(* CODESYS project tcl_simpleunittestlibrary.library
   Company: Red Rock Controls Limited
   Description: ClearTests() added to TTestRunner
   Version: 1.0.7.0
   Placeholder: tcl_SimpleUnitTestLibrary
   Author: Roger Christopher
   Title: tcl_SimpleUnitTestLibrary

Project tree, tasks and I/O mapping:
  libraries: Tc2_EtherCAT, * (Beckhoff Automation GmbH); Tc2_Standard, * (Beckhoff Automation GmbH); Tc2_System, * (Beckhoff Automation GmbH); Tc2_Utilities, * (Beckhoff Automation GmbH); Tc3_DynamicMemory, * (Beckhoff Automation GmbH); Tc3_Module, * (Beckhoff Automation GmbH); tcl_StringUtils, * (Red Rock Controls Limited)
  DUTs/
    data type TTestResult
  GVLs/
    global variables Parameters
    global variables TestFramework
  Unit Test Framework/
    Assertions/
      interface IAssertionMessageList: AddMessage, Clear
      function block TAssertion [ST]: AssertEquals_BLOB, AssertEquals_BOOL, AssertEquals_BYTE, AssertEquals_DINT, AssertEquals_DWORD, AssertEquals_INT, AssertEquals_INTERFACE, AssertEquals_LINT, AssertEquals_LREAL, AssertEquals_PVOID, AssertEquals_REAL, AssertEquals_STRING, AssertEquals_UDINT, AssertEquals_UINT, AssertEquals_ULINT, AssertEquals_WORD, FB_init, AssertionFailed, AssertionMessage
    Message list/
      function block TAssertionMessageList [ST]: AddMessage, Clear
    Test Runner/
      Test Runner/
        function block TTestRunner [ST]: AddTest, AddTestSuite, ClearResults, ClearTests, getTimeStampAsString, Results, TestCount, TestsRunning
    TestSuite/
      interface ITestSuite: AddTest, GetTest, Name, TestCount
      function block TTestSuite [ST]: AddTest, FB_init, GetTest, Name, TestCount
    Unit Test/
      interface IAssertionListener: OnAssertionFailed, TestName
      interface IUnitTest: Execute, Initialise, TestHasFailed, TestHasFinished, TestName
      function block TUnitTestBase [ST]: Execute, FB_init, Initialise, OnAssertionFailed, setTestName, TestFinished, TestHasFailed, TestHasFinished, TestName
  Version/
    global variables Global_Version
  VISUs/
    visualisation Visualization
  GlobalImagePool
  00000000-0000-0000-0000-000000000000|Images\Failed.png
  00000000-0000-0000-0000-000000000000|Images\Passed.png
  00000000-0000-0000-0000-000000000000|Images\BlueRight.png
  text list GlobalTextList
*)

// DUTs/TTestResult
TYPE TTestResult :
STRUCT
    TestName         : T_MaxString;
    TestState        : T_MaxString;
    ImageRef         : T_MaxString;
    TestCompleteTime : T_MaxString;
END_STRUCT
END_TYPE

// GVLs/Parameters
VAR_GLOBAL CONSTANT
    MAX_TESTS              : DINT := 200;
    MAX_ASSERTION_MESSAGES : DINT := 200;
END_VAR

// GVLs/TestFramework
{attribute 'qualified_only'}
VAR_GLOBAL
    TestRunner : TTestRunner;
END_VAR

// Version/Global_Version
{attribute 'TcGenerated'}
{attribute 'no-analysis'}
{attribute 'linkalways'}
// This function has been automatically generated from the project information.
VAR_GLOBAL CONSTANT
	{attribute 'const_non_replaced'}
	stLibVersion_tcl_SimpleUnitTestLibrary : ST_LibVersion := (iMajor := 1, iMinor := 0, iBuild := 7, iRevision := 0, nFlags := 0, sVersion := '1.0.7.0');
END_VAR

// Unit Test Framework/Assertions/IAssertionMessageList
INTERFACE IAssertionMessageList

METHOD AddMessage : BOOL
VAR_INPUT
    Message : T_MaxString;
END_VAR
END_METHOD

METHOD Clear
VAR_INPUT
END_VAR
END_METHOD

END_INTERFACE

// Unit Test Framework/Assertions/TAssertion
FUNCTION_BLOCK TAssertion
VAR_INPUT
END_VAR
VAR_OUTPUT
END_VAR
VAR
    _AssertionFailed : BOOL;
    _AssertionMessage : T_MaxString;
    _ExpectedAsString : T_MaxString;
    _ActualAsString   : T_MaxString;
    _AssertionListener : IAssertionListener;
END_VAR

METHOD AssertEquals_BLOB
VAR_INPUT
    Expected : ANY;
    Actual   : ANY;
    VariableName : T_MaxString;
END_VAR
IF Expected.diSize <> Actual.diSize THEN
    _AssertionFailed := TRUE;
    _AssertionMessage := F_FormatStringEx2('AssertEquals_BLOB failed in %s: Value "%s"', _AssertionListener.TestName, 'Blob.Size');
    _ExpectedAsString := F_FormatString1('  Expected = %d', F_DINT(Expected.diSize));
    _ActualAsString   := F_FormatString1('  Actual   = %d', F_DINT(Actual.diSize));
    _AssertionListener.OnAssertionFailed(_AssertionMessage,_ExpectedAsString,_ActualAsString);
    
ELSIF Expected.TypeClass <> Actual.TypeClass THEN
    _AssertionFailed := TRUE;
    _AssertionMessage := F_FormatStringEx2('AssertEquals_BLOB failed in %s: Value "%s"', _AssertionListener.TestName, 'Blob.TypeClass');
    _ExpectedAsString := F_FormatStringEx1('  Expected = %s', F_TypeClassToString(Expected.TypeClass));
    _ActualAsString   := F_FormatStringEx1('  Actual   = %s', F_TypeClassToString(Actual.TypeClass));
    _AssertionListener.OnAssertionFailed(_AssertionMessage,_ExpectedAsString,_ActualAsString);
    
ELSIF 
    MEMCMP(
        pBuf1 := Expected.pValue, 
        pBuf2 := Actual.pValue, 
        n     := DINT_TO_UDINT(Actual.diSize)) <> 0
THEN
    _AssertionFailed := TRUE;
    _AssertionMessage := F_FormatStringEx1('AssertEquals_BLOB failed in %s: Contents differ', _AssertionListener.TestName);
    _ExpectedAsString := '';
    _ActualAsString   := '';
    _AssertionListener.OnAssertionFailed(_AssertionMessage,_ExpectedAsString,_ActualAsString);
ELSE
    _AssertionFailed  := FALSE;
    _AssertionMessage := '';
END_IF
END_METHOD

METHOD AssertEquals_BOOL 
VAR_INPUT
    Expected : BOOL;
    Actual   : BOOL;
    VariableName : T_MaxString;
END_VAR
IF Expected <> Actual THEN
    _AssertionFailed  := TRUE;
    _AssertionMessage := F_FormatStringEx2('AssertEquals_BOOL failed in %s: Value "%s"', _AssertionListener.TestName, VariableName);
    _ExpectedAsString := F_FormatStringEx1('  Expected = %s', BOOL_TO_STRING(Expected));
    _ActualAsString   := F_FormatStringEx1('  Actual   = %s', BOOL_TO_STRING(Actual));
    _AssertionListener.OnAssertionFailed(_AssertionMessage,_ExpectedAsString,_ActualAsString);
ELSE
    _AssertionFailed   := FALSE;
    _AssertionMessage  := '';
END_IF
END_METHOD

METHOD AssertEquals_BYTE
VAR_INPUT
    Expected : BYTE;
    Actual   : BYTE;
    VariableName : T_MaxString;
END_VAR
IF Expected <> Actual THEN
    _AssertionFailed := TRUE;
    _AssertionMessage := F_FormatStringEx2('AssertEquals_BYTE failed in %s: Value "%s"', _AssertionListener.TestName, VariableName);
    _ExpectedAsString := F_FormatString1('  Expected = %d', F_BYTE(Expected));
    _ActualAsString   := F_FormatString1('  Actual   = %d', F_BYTE(Actual));
    _AssertionListener.OnAssertionFailed(_AssertionMessage,_ExpectedAsString,_ActualAsString);
ELSE
    _AssertionFailed  := FALSE;
    _AssertionMessage := '';
END_IF
END_METHOD

METHOD AssertEquals_DINT 
VAR_INPUT
    Expected : DINT;
    Actual   : DINT;
    VariableName : T_MaxString;
END_VAR
IF Expected <> Actual THEN
    _AssertionFailed  := TRUE;
    _AssertionMessage := F_FormatStringEx2('AssertEquals_DINT failed in %s: Value "%s"', _AssertionListener.TestName, VariableName);
    _ExpectedAsString := F_FormatString1('  Expected = %d', F_DINT(Expected));
    _ActualAsString   := F_FormatString1('  Actual   = %d', F_DINT(Actual));
    _AssertionListener.OnAssertionFailed(_AssertionMessage,_ExpectedAsString,_ActualAsString);
ELSE
    _AssertionFailed  := FALSE;
    _AssertionMessage := '';
END_IF
END_METHOD

METHOD AssertEquals_DWORD
VAR_INPUT
    Expected : DWORD;
    Actual   : DWORD;
    VariableName : T_MaxString;
END_VAR
IF Expected <> Actual THEN
    _AssertionFailed := TRUE;
    _AssertionMessage := F_FormatStringEx2('AssertEquals_DWORD failed in %s: Value "%s"', _AssertionListener.TestName, VariableName);
    _ExpectedAsString := F_FormatString1('  Expected = %d', F_DWORD(Expected));
    _ActualAsString   := F_FormatString1('  Actual   = %d', F_DWORD(Actual));
    _AssertionListener.OnAssertionFailed(_AssertionMessage,_ExpectedAsString,_ActualAsString);
ELSE
    _AssertionFailed  := FALSE;
    _AssertionMessage := '';
END_IF
END_METHOD

METHOD AssertEquals_INT
VAR_INPUT
    Expected : INT;
    Actual   : INT;
    VariableName : T_MaxString;
END_VAR
IF Expected <> Actual THEN
    _AssertionFailed := TRUE;
    _AssertionMessage := F_FormatStringEx2('AssertEquals_INT failed in %s: Value "%s"', _AssertionListener.TestName, VariableName);
    _ExpectedAsString := F_FormatString1('  Expected = %d', F_INT(Expected));
    _ActualAsString   := F_FormatString1('  Actual   = %d', F_INT(Actual));
    _AssertionListener.OnAssertionFailed(_AssertionMessage,_ExpectedAsString,_ActualAsString);
ELSE
    _AssertionFailed  := FALSE;
    _AssertionMessage := '';
END_IF
END_METHOD

METHOD AssertEquals_INTERFACE 
VAR_INPUT
    Expected : __SYSTEM.IQueryInterface;
    Actual   : __SYSTEM.IQueryInterface;
    VariableName : T_MaxString;
END_VAR
IF Expected <> Actual THEN
    _AssertionFailed  := TRUE;
    _AssertionMessage := F_FormatStringEx2('AssertEquals_INTERFACE failed in %s: Value "%s"', _AssertionListener.TestName, VariableName);
    _ExpectedAsString := '  Interfaces Differ';
    _ActualAsString   := '';
    _AssertionListener.OnAssertionFailed(_AssertionMessage,_ExpectedAsString,_ActualAsString);
ELSE
    _AssertionFailed  := FALSE;
    _AssertionMessage := '';
END_IF
END_METHOD

METHOD AssertEquals_LINT 
VAR_INPUT
    Expected : LINT;
    Actual   : LINT;
    VariableName : T_MaxString;
END_VAR
IF Expected <> Actual THEN
    _AssertionFailed  := TRUE;
    _AssertionMessage := F_FormatStringEx2('AssertEquals_LINT failed in %s: Value "%s"', _AssertionListener.TestName, VariableName);
    _ExpectedAsString := F_FormatString1('  Expected = %d', F_LINT(Expected));
    _ActualAsString   := F_FormatString1('  Actual   = %d', F_LINT(Actual));
    _AssertionListener.OnAssertionFailed(_AssertionMessage,_ExpectedAsString,_ActualAsString);
ELSE
    _AssertionFailed  := FALSE;
    _AssertionMessage := '';
END_IF
END_METHOD

METHOD AssertEquals_LREAL 
VAR_INPUT
    Expected : LREAL;
    Actual   : LREAL;
    Delta    : LREAL;
    VariableName : T_MaxString;
END_VAR
IF ABS(Expected - Actual) >= Delta THEN
    _AssertionFailed  := TRUE;
    _AssertionMessage := F_FormatStringEx2('AssertEquals_LREAL failed in %s: Value "%s"', _AssertionListener.TestName, VariableName);
    _ExpectedAsString := F_FormatString1('  Expected = %f', F_LREAL(Expected));
    _ActualAsString   := F_FormatString1('  Actual   = %f', F_LREAL(Actual));
    _AssertionListener.OnAssertionFailed(_AssertionMessage,_ExpectedAsString,_ActualAsString);
ELSE
    _AssertionFailed  := FALSE;
    _AssertionMessage := '';
END_IF
END_METHOD

METHOD AssertEquals_PVOID 
VAR_INPUT
    Expected : PVOID;
    Actual   : PVOID;
    VariableName : T_MaxString;
END_VAR
IF Expected <> Actual THEN
    _AssertionFailed  := TRUE;
    _AssertionMessage := F_FormatStringEx2('AssertEquals_PVOID failed in %s: Value "%s"', _AssertionListener.TestName, VariableName);
    _ExpectedAsString := F_FormatString1('  Expected = %d', F_PVOID(Expected));
    _ActualAsString   := F_FormatString1('  Actual   = %d', F_PVOID(Actual));
    _AssertionListener.OnAssertionFailed(_AssertionMessage,_ExpectedAsString,_ActualAsString);
ELSE
    _AssertionFailed  := FALSE;
    _AssertionMessage := '';
END_IF
END_METHOD

METHOD AssertEquals_REAL 
VAR_INPUT
    Expected : REAL;
    Actual   : REAL;
    Delta    : REAL;
    VariableName : T_MaxString;
END_VAR
IF ABS(Expected - Actual) >= Delta THEN
    _AssertionFailed  := TRUE;
    _AssertionMessage := F_FormatStringEx2('AssertEquals_REAL failed in %s: Value "%s"', _AssertionListener.TestName, VariableName);
    _ExpectedAsString := F_FormatString1('  Expected = %f', F_REAL(Expected));
    _ActualAsString   := F_FormatString1('  Actual   = %f', F_REAL(Actual));
    _AssertionListener.OnAssertionFailed(_AssertionMessage,_ExpectedAsString,_ActualAsString);
ELSE
    _AssertionFailed  := FALSE;
    _AssertionMessage := '';
END_IF
END_METHOD

METHOD AssertEquals_STRING
VAR_INPUT
    Expected : T_MaxString;
    Actual   : T_MaxString;
    VariableName : T_MaxString;
END_VAR
IF Expected <> Actual THEN
    _AssertionFailed := TRUE;
    _AssertionMessage := F_FormatStringEx2('AssertEquals_STRING failed in %s: Value "%s"', _AssertionListener.TestName, VariableName);
    _ExpectedAsString := F_FormatStringEx1('  Expected = %s', Expected);
    _ActualAsString   := F_FormatStringEx1('  Actual   = %s', Actual);
    _AssertionListener.OnAssertionFailed(_AssertionMessage,_ExpectedAsString,_ActualAsString);
ELSE
    _AssertionFailed   := FALSE;
    _AssertionMessage  := '';
    _ExpectedAsString  := '';
    _ActualAsString    := '';
END_IF
END_METHOD

METHOD AssertEquals_UDINT
VAR_INPUT
    Expected : UDINT;
    Actual   : UDINT;
    VariableName : T_MaxString;
END_VAR
IF Expected <> Actual THEN
    _AssertionFailed := TRUE;
    _AssertionMessage := F_FormatStringEx2('AssertEquals_UDINT failed in %s: Value "%s"', _AssertionListener.TestName, VariableName);
    _ExpectedAsString := F_FormatString1('  Expected = %d', F_UDINT(Expected));
    _ActualAsString   := F_FormatString1('  Actual   = %d', F_UDINT(Actual));
    _AssertionListener.OnAssertionFailed(_AssertionMessage,_ExpectedAsString,_ActualAsString);
ELSE
    _AssertionFailed  := FALSE;
    _AssertionMessage := '';
END_IF
END_METHOD

METHOD AssertEquals_UINT
VAR_INPUT
    Expected : UINT;
    Actual   : UINT;
    VariableName : T_MaxString;
END_VAR
IF Expected <> Actual THEN
    _AssertionFailed := TRUE;
    _AssertionMessage := F_FormatStringEx2('AssertEquals_UINT failed in %s: Value "%s"', _AssertionListener.TestName, VariableName);
    _ExpectedAsString := F_FormatString1('  Expected = %d', F_UINT(Expected));
    _ActualAsString   := F_FormatString1('  Actual   = %d', F_UINT(Actual));
    _AssertionListener.OnAssertionFailed(_AssertionMessage,_ExpectedAsString,_ActualAsString);
ELSE
    _AssertionFailed  := FALSE;
    _AssertionMessage := '';
END_IF
END_METHOD

METHOD AssertEquals_ULINT 
VAR_INPUT
    Expected : ULINT;
    Actual   : ULINT;
    VariableName : T_MaxString;
END_VAR
IF Expected <> Actual THEN
    _AssertionFailed  := TRUE;
    _AssertionMessage := F_FormatStringEx2('AssertEquals_ULINT failed in %s: Value "%s"', _AssertionListener.TestName, VariableName);
    _ExpectedAsString := F_FormatString1('  Expected = %d', F_ULINT(Expected));
    _ActualAsString   := F_FormatString1('  Actual   = %d', F_ULINT(Actual));
    _AssertionListener.OnAssertionFailed(_AssertionMessage,_ExpectedAsString,_ActualAsString);
ELSE
    _AssertionFailed  := FALSE;
    _AssertionMessage := '';
END_IF
END_METHOD

METHOD AssertEquals_WORD
VAR_INPUT
    Expected : WORD;
    Actual   : WORD;
    VariableName : T_MaxString;
END_VAR
IF Expected <> Actual THEN
    _AssertionFailed := TRUE;
    _AssertionMessage := F_FormatStringEx2('AssertEquals_WORD failed in %s: Value "%s"', _AssertionListener.TestName, VariableName);
    _ExpectedAsString := F_FormatString1('  Expected = %d', F_WORD(Expected));
    _ActualAsString   := F_FormatString1('  Actual   = %d', F_WORD(Actual));
    _AssertionListener.OnAssertionFailed(_AssertionMessage,_ExpectedAsString,_ActualAsString);
ELSE
    _AssertionFailed  := FALSE;
    _AssertionMessage := '';
END_IF
END_METHOD

METHOD FB_init : BOOL
VAR_INPUT
	bInitRetains : BOOL; // if TRUE, the retain variables are initialized (warm start / cold start)
	bInCopyCode : BOOL;  // if TRUE, the instance afterwards gets moved into the copy code (online change)
    AssertionListener : IAssertionListener;
END_VAR
_AssertionListener := AssertionListener;
END_METHOD

PROPERTY AssertionFailed : BOOL
GET
AssertionFailed := _AssertionFailed;
END_GET
END_PROPERTY

PROPERTY AssertionMessage : T_MaxString
GET
AssertionMessage := _AssertionMessage;
END_GET
END_PROPERTY

END_FUNCTION_BLOCK

// Unit Test Framework/Unit Test/IAssertionListener
INTERFACE IAssertionListener

METHOD OnAssertionFailed
VAR_INPUT
    AssertionMessage : T_MaxString;
    ExpectedAsString : T_MaxString;
    ActualAsString   : T_MaxString;
END_VAR
END_METHOD

PROPERTY TestName : T_MaxString
GET
END_GET
END_PROPERTY

END_INTERFACE

// Unit Test Framework/Message list/TAssertionMessageList
FUNCTION_BLOCK TAssertionMessageList IMPLEMENTS IAssertionMessageList
VAR
    _Messages : ARRAY[0..MAX_ASSERTION_MESSAGES] OF T_MaxString;
    _Count : INT;
END_VAR

METHOD AddMessage : BOOL
VAR_INPUT
    Message : T_MaxString;
END_VAR
IF _Count <= MAX_ASSERTION_MESSAGES THEN
    _Messages[_Count] := Message;
    _Count := _Count + 1;
    AddMessage := TRUE;
END_IF
END_METHOD

METHOD Clear
VAR_INPUT
END_VAR
MEMSET(
    destAddr := ADR(_Messages), 
    fillByte := 0, 
    n        := SIZEOF(_Messages));
_Count := 0;
END_METHOD

END_FUNCTION_BLOCK

// Unit Test Framework/Test Runner/Test Runner/TTestRunner
FUNCTION_BLOCK TTestRunner 
VAR_INPUT
    RunTestsSequentially : BOOL := TRUE; 
    ManualTestRunsOnly   : BOOL := TRUE; // Set true to enforce "Manual run only"
END_VAR
VAR
    Run : BOOL := TRUE;
    
    State :(
        PreInit,
        Init,
        RunTests_Concurrently,
        RunTests_Sequentially,
        CheckResults);
        
    i : INT;
    CompletedTestsCount : INT;
    FailedTestsCount : INT;
    CurrentTestIndex : INT;
    
    _TestsRunning : BOOL;
    _Results : T_MaxString;
    _AllTestsCompleted : BOOL;
    _TestCount : INT;
    
    Tests : ARRAY[0..MAX_TESTS] OF IUnitTest;
    TestResults : ARRAY[0..MAX_TESTS] OF TTestResult;
    AssertionMessages : TAssertionMessageList;
    
    TestsCompletedPercentage : LREAL;
END_VAR

CASE State OF
    PreInit:
        Run := NOT ManualTestRunsOnly;
        State := Init;
    Init:
        IF Run THEN
            Run := FALSE;
            ClearResults();
            AssertionMessages.Clear();
            FOR i := 0 TO _TestCount - 1 DO
                IF Tests[i] <> 0 THEN
                    Tests[i].Initialise(AssertionMessages);
				END_IF
			END_FOR
            _TestsRunning := TRUE;
            IF RunTestsSequentially THEN
                CurrentTestIndex := 0;
                State := RunTests_Sequentially;
            ELSE
                State := RunTests_Concurrently;
            END_IF
		END_IF
        
    RunTests_Concurrently:
        CompletedTestsCount := 0;
        FOR i := 0 TO _TestCount - 1 DO
            IF Tests[i] <> 0 THEN
                IF Tests[i].TestHasFinished THEN
                    TestResults[i].TestCompleteTime := getTimeStampAsString();
                    IF Tests[i].TestHasFailed THEN
                        TestResults[i].TestName  := Tests[i].TestName;
                        TestResults[i].TestState := 'Failed';
                        TestResults[i].ImageRef  := '3';
                        FailedTestsCount := FailedTestsCount + 1;
                    ELSE
                        TestResults[i].TestName  := Tests[i].TestName;
                        TestResults[i].TestState := 'Passed';
                        TestResults[i].ImageRef  := '2';
                    END_IF    
                    
                    CompletedTestsCount := CompletedTestsCount + 1;
                    TestsCompletedPercentage := CompletedTestsCount * 100/_TestCount;
                    _Results := F_FormatString2('%d Tests completed, %d Tests Failed',F_INT(CompletedTestsCount),F_INT(FailedTestsCount));
                ELSE
                    TestResults[i].TestName  := Tests[i].TestName;
                    TestResults[i].TestState := 'Running';
                    TestResults[i].ImageRef  := '1';
                    Tests[i].Execute();
                END_IF
            END_IF
        END_FOR
        IF CompletedTestsCount >= _TestCount THEN
            State := CheckResults;
		END_IF
        
    RunTests_Sequentially:
        IF Tests[CurrentTestIndex] <> 0 THEN
            IF Tests[CurrentTestIndex].TestHasFinished THEN
                TestResults[CurrentTestIndex].TestCompleteTime := getTimeStampAsString();
                IF Tests[CurrentTestIndex].TestHasFailed THEN
                    TestResults[CurrentTestIndex].TestName  := Tests[CurrentTestIndex].TestName;
                    TestResults[CurrentTestIndex].TestState := 'Failed';
                    TestResults[CurrentTestIndex].ImageRef  := '3';
                    FailedTestsCount := FailedTestsCount + 1;
                ELSE
                    TestResults[CurrentTestIndex].TestName  := Tests[CurrentTestIndex].TestName;
                    TestResults[CurrentTestIndex].TestState := 'Passed';
                    TestResults[CurrentTestIndex].ImageRef  := '2';
                END_IF    
                
                CompletedTestsCount := CompletedTestsCount + 1;
                CurrentTestIndex := CurrentTestIndex + 1;
                TestsCompletedPercentage := CompletedTestsCount * 100/_TestCount;
                _Results := F_FormatString2('%d Tests completed, %d Tests Failed',F_INT(CompletedTestsCount),F_INT(FailedTestsCount));
            ELSE
                TestResults[CurrentTestIndex].TestName  := Tests[CurrentTestIndex].TestName;
                TestResults[CurrentTestIndex].TestState := 'Running';
                TestResults[CurrentTestIndex].ImageRef  := '1';
                Tests[CurrentTestIndex].Execute();
            END_IF
        END_IF

        IF CompletedTestsCount >= _TestCount THEN
            State := CheckResults;
		END_IF

    CheckResults:
        _Results := F_FormatString2('%d Tests completed, %d Tests Failed',F_INT(CompletedTestsCount),F_INT(FailedTestsCount));
        _TestsRunning := FALSE;
        _AllTestsCompleted := TRUE;
        
        State := Init;
    
    
END_CASE

METHOD AddTest : BOOL
VAR_INPUT
    UnitTest : IUnitTest;
END_VAR
IF _TestCount < MAX_TESTS THEN
    Tests[_TestCount] := UnitTest;
    _TestCount := _TestCount + 1;
    AddTest := TRUE;
ELSE
    AssertionMessages.AddMessage('Maximum unit tests exceeded!');
END_IF
END_METHOD

METHOD AddTestSuite : BOOL
VAR_INPUT
    TestSuite : ITestSuite;
END_VAR
VAR
    i : INT;
    UnitTestToAdd : IUnitTest;
END_VAR
IF TestSuite.TestCount > 0 THEN
    FOR i := 0 TO TestSuite.TestCount - 1 DO
        UnitTestToAdd := TestSuite.GetTest(i);
        AddTest(UnitTestToAdd);
    END_FOR
END_IF
END_METHOD

METHOD ClearResults
VAR_INPUT
END_VAR
_Results := '';
_AllTestsCompleted := FALSE;
FailedTestsCount := 0;
CompletedTestsCount := 0;
TestsCompletedPercentage := 0;

MEMSET(
    destAddr := ADR(TestResults), 
    fillByte := 0, 
    n        := SIZEOF(TestResults));
END_METHOD

METHOD ClearTests
VAR_INPUT
END_VAR
MEMSET(
    destAddr := ADR(Tests),
    fillByte := 0,
    n        := SIZEOF(Tests));
_TestCount := 0;
END_METHOD

METHOD PRIVATE getTimeStampAsString : T_MaxString
VAR
	CurrentDcTime : T_DCTIME64;
    Now : TIMESTRUCT;
END_VAR
CurrentDcTime := F_GetActualDcTime64();
Now := DCTIME64_TO_SYSTEMTIME(CurrentDcTime);
getTimeStampAsString := tcl_StringUtils.F_TimeAsString_ms(Now);
END_METHOD

PROPERTY Results : T_MaxString
GET
Results := _Results;
END_GET
END_PROPERTY

PROPERTY TestCount : INT
GET
TestCount := _TestCount;
END_GET
END_PROPERTY

PROPERTY TestsRunning : BOOL
GET
TestsRunning := _TestsRunning;
END_GET
END_PROPERTY

END_FUNCTION_BLOCK

// Unit Test Framework/Unit Test/IUnitTest
INTERFACE IUnitTest EXTENDS __SYSTEM.IQueryInterface

METHOD Execute
END_METHOD

METHOD Initialise
VAR_INPUT
    MessageList : IAssertionMessageList;
END_VAR
END_METHOD

PROPERTY TestHasFailed : BOOL
GET
END_GET
END_PROPERTY

PROPERTY TestHasFinished : BOOL
GET
END_GET
END_PROPERTY

PROPERTY TestName : T_MaxString
GET
END_GET
END_PROPERTY

END_INTERFACE

// Unit Test Framework/TestSuite/ITestSuite
INTERFACE ITestSuite

METHOD AddTest : BOOL
VAR_INPUT
    UnitTest : IUnitTest;
END_VAR
END_METHOD

METHOD GetTest : IUnitTest
VAR_INPUT
    Index : INT;
END_VAR
END_METHOD

PROPERTY Name : T_MaxString
GET
END_GET
END_PROPERTY

PROPERTY TestCount : INT
GET
END_GET
END_PROPERTY

END_INTERFACE

// Unit Test Framework/TestSuite/TTestSuite
{attribute 'reflection'}
FUNCTION_BLOCK TTestSuite IMPLEMENTS ITestSuite
VAR_INPUT
END_VAR
VAR_OUTPUT
END_VAR
VAR
    {attribute 'instance-path'} 
    {attribute 'no_init'}
    _TestSuiteName       : T_MaxString; // Automatically initialised with the full name of the instance
    _TestCount : INT;
    Tests : ARRAY[0..MAX_TESTS_PER_TEST_SUITE] OF IUnitTest;
END_VAR
VAR CONSTANT
    MAX_TESTS_PER_TEST_SUITE              : DINT := 100;
END_VAR

METHOD AddTest : BOOL
VAR_INPUT
    UnitTest : IUnitTest;
END_VAR
IF _TestCount < MAX_TESTS_PER_TEST_SUITE THEN
    Tests[_TestCount] := UnitTest;
    _TestCount := _TestCount + 1;
    AddTest := TRUE;
END_IF
END_METHOD

METHOD FB_init : BOOL
VAR_INPUT
	bInitRetains : BOOL; // if TRUE, the retain variables are initialized (warm start / cold start)
	bInCopyCode : BOOL;  // if TRUE, the instance afterwards gets moved into the copy code (online change)
END_VAR
VAR
    StringSplitter : TStringSplitter;
END_VAR
StringSplitter.Init(
    Str := _TestSuiteName,
    Delim1 := '.',
    Delim2 := '');
    
WHILE StringSplitter.HasMore() DO
    _TestSuiteName := StringSplitter.GetNext(); // to get last sub-section
END_WHILE
END_METHOD

METHOD GetTest : IUnitTest
VAR_INPUT
    Index : INT;
END_VAR
IF Index >= 0 AND Index < _TestCount THEN
    GetTest := Tests[Index];
END_IF
END_METHOD

PROPERTY Name : T_MaxString
GET
Name := _TestSuiteName;
END_GET
END_PROPERTY

PROPERTY TestCount : INT
GET
TestCount := _TestCount;
END_GET
END_PROPERTY

END_FUNCTION_BLOCK

// Unit Test Framework/Unit Test/TUnitTestBase
{attribute 'reflection'}
FUNCTION_BLOCK ABSTRACT TUnitTestBase IMPLEMENTS IUnitTest, IAssertionListener
VAR
    {attribute 'instance-path'} 
    {attribute 'no_init'}
    _TestName       : T_MaxString; // Automatically initialised with the full name of the instance
    _TestFailed     : BOOL;
    _TestFinished   : BOOL;
    _ImageRef       : STRING;
    _MessageList    : IAssertionMessageList;
    
    Assertion : TAssertion(AssertionListener := THIS^); // Callback to allow the Assertion to update the message list on assertion failed

END_VAR

METHOD Execute
THIS^();
END_METHOD

METHOD FB_init : BOOL
VAR_INPUT
	bInitRetains : BOOL; // if TRUE, the retain variables are initialized (warm start / cold start)
	bInCopyCode : BOOL;  // if TRUE, the instance afterwards gets moved into the copy code (online change)
    TestSuite : ITestSuite;
END_VAR
IF TestSuite <> 0 THEN
    THIS^.setTestName(TestSuite.Name);
    TestSuite.AddTest(THIS^);
END_IF
END_METHOD

METHOD Initialise
VAR_INPUT
    MessageList : IAssertionMessageList;
END_VAR
_TestFailed   := FALSE;
_TestFinished := FALSE;
_ImageRef     := '0';
_MessageList  := MessageList;
END_METHOD

METHOD OnAssertionFailed
VAR_INPUT
    AssertionMessage : T_MaxString;
    ExpectedAsString : T_MaxString;
    ActualAsString   : T_MaxString;
END_VAR
_TestFailed := TRUE;
_MessageList.AddMessage(AssertionMessage);

IF ExpectedAsString <> '' THEN
    _MessageList.AddMessage(ExpectedAsString);
END_IF

IF ActualAsString <> '' THEN
    _MessageList.AddMessage(ActualAsString);
END_IF
END_METHOD

METHOD setTestName
VAR_INPUT
    GroupName : STRING;
END_VAR
VAR
    StringSplitter : TStringSplitter;
END_VAR
StringSplitter.Init(
    Str := _TestName,
    Delim1 := '.',
    Delim2 := '');
    
WHILE StringSplitter.HasMore() DO
    _TestName := StringSplitter.GetNext(); // to get last sub-section
END_WHILE

IF GroupName <> '' THEN
    _TestName := F_FormatStringEx2(Format := '%s.%s',arg1 := GroupName, arg2 := _TestName);
END_IF
END_METHOD

METHOD TestFinished
VAR_INPUT
END_VAR
_TestFinished := TRUE;
END_METHOD

PROPERTY TestHasFailed : BOOL
GET
TestHasFailed := _TestFailed;
END_GET
END_PROPERTY

PROPERTY TestHasFinished : BOOL
GET
TestHasFinished := _TestFinished;
END_GET
END_PROPERTY

PROPERTY TestName : T_MaxString
GET
TestName := _TestName;
END_GET
END_PROPERTY

END_FUNCTION_BLOCK

// VISUs/Visualization
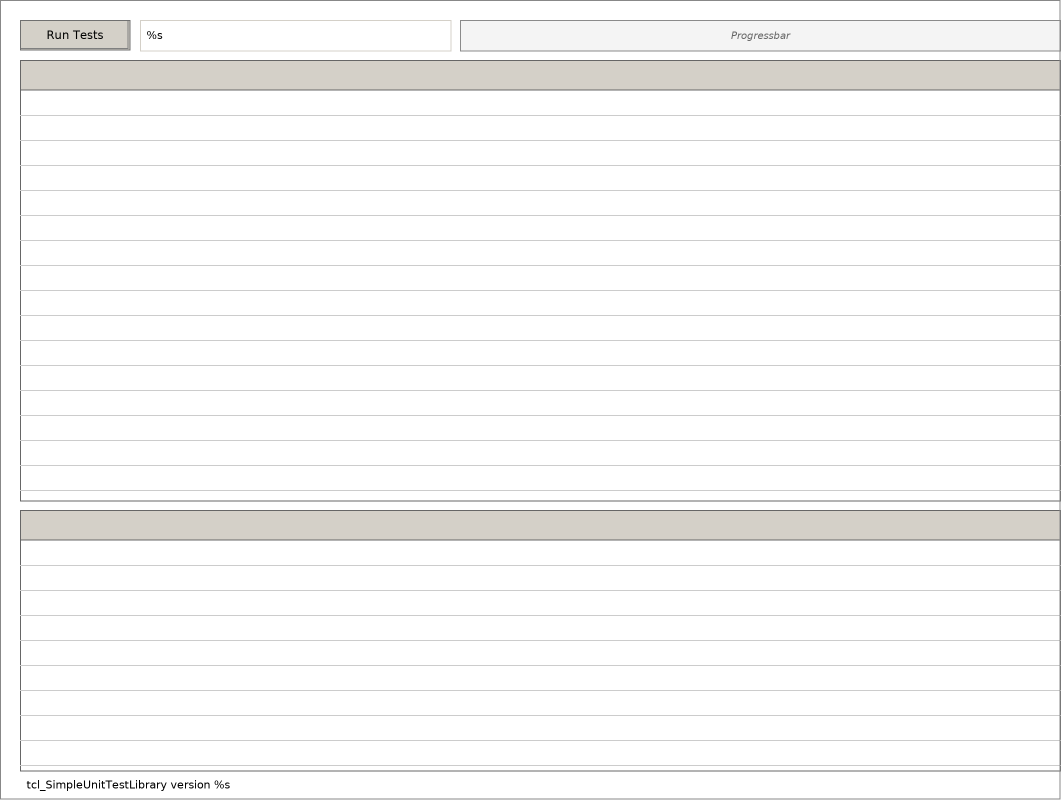
VISUALIZATION Visualization  // 1061x800
    Button (20,20 110x30), "Run Tests"
        tap TestFramework.TestRunner.Run
    Textfield (140,20 311x31), "%s", text variable: TestFramework.TestRunner._Results
    Table (20,60 1041x441), data array: TestFramework.TestRunner.TestResults
        p2170511999: TestFramework.TestRunner.TestResults[INDEX].ImageRef
        p1755163831: Test State
        p338671338: TestFramework.TestRunner.TestResults[INDEX].TestState
        p511219082: Test Name
        p1892666644: TestFramework.TestRunner.TestResults[INDEX].TestName
        p2232123230: Time
        p3854506369: TestFramework.TestRunner.TestResults[INDEX].TestCompleteTime
    Table (20,510 1041x261), data array: TestFramework.TestRunner.AssertionMessages._Messages
        p3854506369: TestFramework.TestRunner.AssertionMessages._Messages[INDEX]
        p2232123230: Assertion Messages
    Progressbar (460,20 601x31), variable: TestFramework.TestRunner.TestsCompletedPercentage
    Rectangle (20,770 650x30), "tcl_SimpleUnitTestLibrary version %s", text variable: Global_Version.stLibVersion_tcl_SimpleUnitTestLibrary.sVersion
END_VISUALIZATION
